(* PLC project op_door, Dassault Systèmes ControlBuild 2024x *)
(* stored: creationDateTime 2023-10-03T11:13:48-01:00 *)

FUNCTION_BLOCK tni_train.op_door
  VAR_INPUT
    compressedAir : REAL := 200.0;
    cmdSupply : BOOL := true;
    sensorSupply : BOOL := true;
  END_VAR
  VAR_INPUT
    openDoorCmd : BOOL := false;
    closeDoorCmd : BOOL := false;
  END_VAR
  VAR_INPUT
    lockActive : BOOL := false;
  END_VAR
  VAR_OUTPUT
    doorOpened : BOOL := false;
    doorClosed : BOOL := false;
  END_VAR
  VAR
    increment : REAL := 0.0;
    openDoor : BOOL := false;
    closeDoor : BOOL := false;
    doorPosition : REAL := 0.0;
  END_VAR
  VAR CONSTANT
    length : REAL := 1000.0;
    doorClosedSensorLogic : BOOL := true;
    doorOpenedSensorLogic : BOOL := true;
  END_VAR
  VAR
    d_locking : BOOL := false;
    v_d_locking : REAL := 50.0;
    d_doorClosedSensor : BOOL := false;
    v_d_doorClosedSensor : BOOL := false;
    d_doorOpenedSensor : BOOL := false;
    v_d_doorOpenedSensor : BOOL := false;
  END_VAR

(* -----------------------------------------------------------------	*)
(* Type : Model of Operative Behaviour					*)
(* Category :  Sample application TNI train				*)
(* Author : Franck Corbier Techniques Nouvelles d'Informatique	*)
(* Update date : October 2002						*)
(* -----------------------------------------------------------------	*)

(* -----------------------------------------------------------------	*)
(* Management of the door's movement					*)
(* -----------------------------------------------------------------	*)
IF (d_locking) THEN increment := 0.0;
ELSE
	increment := compressedAir * (CLOCK_PERIOD/1000000);
	IF (cmdSupply) THEN
		IF (openDoorCmd AND NOT closeDoorCmd) THEN
			openDoor := TRUE;
			closeDoor := FALSE;
		END_IF;
		IF ( NOT openDoorCmd AND closeDoorCmd) THEN 
			openDoor := FALSE;
			closeDoor := TRUE;
		END_IF;
	END_IF;
	IF (openDoor) THEN
		IF ( doorPosition < length) THEN doorPosition := doorPosition + increment; END_IF;
		IF ( doorPosition > length) THEN doorPosition := length; END_IF;
	END_IF;
	IF (closeDoor) THEN 
		IF ( doorPosition > 0.0 ) THEN doorPosition := doorPosition - increment; END_IF;
		IF ( doorPosition < 0.0 ) THEN doorPosition := 0.0; END_IF;
	END_IF;
END_IF;


(* -----------------------------------------------------------------	*)
(* Management of the sensors' state					*)
(* -----------------------------------------------------------------	*)
IF (d_doorOpenedSensor) THEN doorOpened := v_d_doorOpenedSensor;
ELSE
	IF (sensorSupply) THEN doorOpened := (doorPosition >= length) XOR NOT doorOpenedSensorLogic;
	ELSE doorOpened := FALSE;
	END_IF;
END_IF;

IF (d_doorClosedSensor) THEN doorClosed := v_d_doorClosedSensor;
ELSE
	IF (sensorSupply) THEN doorClosed := (doorPosition <= 0.0) XOR NOT doorClosedSensorLogic;
  	ELSE doorClosed := FALSE;
	END_IF;
END_IF;
END_FUNCTION_BLOCK
